TYPE ST_PIEZO_AXIS_REF :
STRUCT
END_STRUCT
END_TYPE

(* stored: Version 1.1.0.1
   DUT ST_PIEZO_AXIS_REF: Id {45df8925-8963-45e1-a409-9fa648718788} *)
